Fanuc TP program (LS listing): A_SOUNDL.LS

/PROG  A_SOUNDL
/ATTR
OWNER		= MNEDITOR;
COMMENT		= "SOUND 1sec";
PROG_SIZE	= 202;
CREATE		= DATE 22-01-21  TIME 13:38:20;
MODIFIED	= DATE 22-02-02  TIME 11:06:54;
FILE_NAME	= A_SOUNDL;
VERSION		= 0;
LINE_COUNT	= 2;
MEMORY_SIZE	= 566;
PROTECT		= READ_WRITE;
TCD:  STACK_SIZE	= 0,
      TASK_PRIORITY	= 50,
      TIME_SLICE	= 0,
      BUSY_LAMP_OFF	= 0,
      ABORT_REQUEST	= 0,
      PAUSE_REQUEST	= 0;
DEFAULT_GROUP	= 1,*,*,*,*;
CONTROL_CODE	= 00000000 00000000;
/APPL
/MN
   1:  DO[10:table1 ring]=PULSE,1.0sec ;
   2:  DO[13:table2 ring]=PULSE,1.0sec ;
/POS
/END
